FUNCTION TryConvert_BOOL_TO_TIME : BOOL
VAR_INPUT
	in : BOOL;
	out : REFERENCE TO TIME;
END_VAR

out := BOOL_TO_TIME(in);
TryConvert_BOOL_TO_TIME := TRUE;

END_FUNCTION

(* stored: Version 1.1.0.1, ProductVersion 3.1.4024.12
   POU TryConvert_BOOL_TO_TIME: Id {70a79800-97a1-448f-ba0d-0737734a8af9}, SpecialFunc None *)
